{attribute 'GeneratedUsingTerminal: ER3204-0002-0021'}
{attribute addProperty BoxType "ER3204-0002-0021"}
{attribute addProperty Id "UnderrangeBOOL1OverrangeBOOL1Limit_1BYTE1Limit_2BYTE1ErrorBOOL1TxPDO_StateBOOL1TxPDO_ToggleBOOL1"}
{attribute addProperty CRC "4073614737"}
{attribute addProperty Size "7"}
TYPE Status_F2CE6D91 :
STRUCT
	{attribute addProperty Name "Underrange"}
	Underrange : BOOL;
	{attribute addProperty Name "Overrange"}
	Overrange : BOOL;
	{attribute addProperty Name "Limit_1"}
	Limit_1 : BYTE;
	{attribute addProperty Name "Limit_2"}
	Limit_2 : BYTE;
	{attribute addProperty Name "Error"}
	Error : BOOL;
	{attribute addProperty Name "TxPDO_State"}
	TxPDO_State : BOOL;
	{attribute addProperty Name "TxPDO_Toggle"}
	TxPDO_Toggle : BOOL;
END_STRUCT
END_TYPE

(* stored: Version 1.2.0.0, ProductVersion 3.1.4024.9
   DUT Status_F2CE6D91: Id {2888ea1b-e131-410c-88e0-6c2d66971ccc} *)
